FUNCTION_BLOCK TurntableControl (* Basic FB with empty ECC *)
  (* Standard: 61499-2 *)
  (* Version 1.0, 2021-09-15, dorofeev *)
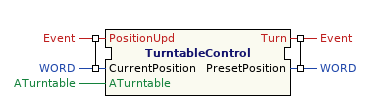
  EVENT_INPUT
    PositionUpd WITH CurrentPosition;
  END_EVENT
  EVENT_OUTPUT
    Turn WITH PresetPosition;
  END_EVENT
  VAR_INPUT
    CurrentPosition : WORD;
  END_VAR
  VAR_OUTPUT
    PresetPosition : WORD;
  END_VAR
  SOCKETS
    ATurntable : ATurntable;
  END_SOCKETS
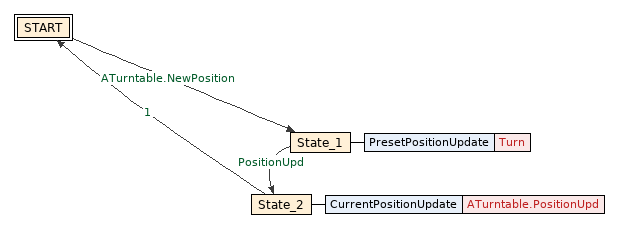
  EC_STATES
    START; (* Initial State *)
    State_1 : PresetPositionUpdate -> Turn;
    State_2 : CurrentPositionUpdate -> ATurntable.PositionUpd;
  END_STATES
  EC_TRANSITIONS
    State_1 TO State_2 := PositionUpd;
    State_2 TO START := 1;
    START TO State_1 := ATurntable.NewPosition;
  END_TRANSITIONS
  ALGORITHM PresetPositionUpdate IN ST: (* New Algorithm *)
PresetPosition := ATurntable.Position;
  END_ALGORITHM
  ALGORITHM CurrentPositionUpdate IN ST: (* New Algorithm *)
ATurntable.CurrentPosition := CurrentPosition;
  END_ALGORITHM
END_FUNCTION_BLOCK
